(* CODESYS project native.xml

Project tree, tasks and I/O mapping:
  Device : CODESYS Control Win V3 x64, CODESYS, version 3.5.21.40
    application Application
      libraries: Standard, 3.5.18.0 (System)
      task MainTask (cyclic, interval t#20ms, priority 1) calls PLC_PRG
      data type E_SystemState
      global variables GVL_IO
      global variables GVL_System
      program PLC_PRG [ST]
*)

// Device/Application/E_SystemState
TYPE E_SystemState :
(
    STOPPED,
    IDLE_READY,
    WAIT_TRAY_EMPTY,
    TRANSFER,
    FAULT
);
END_TYPE

// Device/Application/GVL_IO
{attribute 'qualified_only'}
VAR_GLOBAL
	 (* Inputs *)
    PB_START       : BOOL;
    PB_STOP        : BOOL;
    PB_RESET       : BOOL;
    E_STOP_OK      : BOOL := TRUE;

    PE_INFEED      : BOOL;
    PE_CLEAR       : BOOL := TRUE;    (* often 'clear' is TRUE when not blocked *)

    ITEM_TYPE_A    : BOOL;            (* TRUE = route to Tray A *)
    TRAY_A_EMPTY   : BOOL := TRUE;
    TRAY_B_EMPTY   : BOOL := TRUE;

    (* Outputs *)
    MTR_RUN        : BOOL;
    DIVERT_TO_A    : BOOL;
    DIVERT_TO_B    : BOOL;
    ALARM          : BOOL;
END_VAR

// Device/Application/GVL_System
{attribute 'qualified_only'}
VAR_GLOBAL
	State			: E_SystemState := STOPPED;
	NextState		: E_SystemState := STOPPED;
	
	RouteToA     : BOOL;          (* latched route for current item *)
    RouteLatched : BOOL := FALSE; (* true once route is captured *)
    FaultLatched : BOOL := FALSE;

    Prev_PE_Clear : BOOL := TRUE; (* for edge detect *)
END_VAR

// Device/Application/PLC_PRG
PROGRAM PLC_PRG
VAR
	  clear_rise : BOOL;
END_VAR

(* Default: remain in current state *)
GVL_System.NextState := GVL_System.State;

(* Rising edge when PE_CLEAR goes from 0 -> 1 (blocked -> clear) *)
clear_rise := (NOT GVL_System.Prev_PE_Clear) AND (GVL_IO.PE_CLEAR);
GVL_System.Prev_PE_Clear := GVL_IO.PE_CLEAR;

(* Default outputs: safe *)
GVL_IO.MTR_RUN := FALSE;
GVL_IO.DIVERT_TO_A := FALSE;
GVL_IO.DIVERT_TO_B := FALSE;
GVL_IO.ALARM := FALSE;

(* E-stop fault: immediate, latched *)
IF NOT GVL_IO.E_STOP_OK THEN
    GVL_System.FaultLatched := TRUE;
    GVL_System.State := FAULT;
    RETURN;
END_IF;

CASE GVL_System.State OF

STOPPED:
    (* System is safe, waiting for start *)
	
	GVL_System.RouteLatched := FALSE;
	
    IF GVL_IO.PB_START AND NOT GVL_System.FaultLatched THEN
        GVL_System.NextState := IDLE_READY;
    END_IF;

IDLE_READY:
    (* waiting for item *)
    IF GVL_IO.PE_INFEED THEN
        GVL_System.NextState := WAIT_TRAY_EMPTY;
    END_IF;

WAIT_TRAY_EMPTY:
    (* Latch route once per item *)
    IF NOT GVL_System.RouteLatched THEN
        GVL_System.RouteToA := GVL_IO.ITEM_TYPE_A;   (* TRUE=A, FALSE=B *)
        GVL_System.RouteLatched := TRUE;
    END_IF;

    (* Wait until destination tray is empty *)
    IF GVL_System.RouteToA THEN
        (* Route A *)
        IF GVL_IO.TRAY_A_EMPTY THEN
            GVL_System.NextState := TRANSFER;
        END_IF;
    ELSE
        (* Route B *)
        IF GVL_IO.TRAY_B_EMPTY THEN
            GVL_System.NextState := TRANSFER;
        END_IF;
    END_IF;

TRANSFER:
    (* Command diverter to latched route *)
    IF GVL_System.RouteToA THEN
        GVL_IO.DIVERT_TO_A := TRUE;
    ELSE
        GVL_IO.DIVERT_TO_B := TRUE;
    END_IF;

    (* Run conveyor *)
    GVL_IO.MTR_RUN := TRUE;

    (* Stop transfer when item clears the zone *)
    IF clear_rise THEN
        GVL_IO.MTR_RUN := FALSE;
        GVL_System.RouteLatched := FALSE;     (* ready for next item *)
        GVL_System.NextState := IDLE_READY;
    END_IF;

FAULT:
    GVL_IO.ALARM := TRUE;
    IF GVL_IO.PB_RESET AND GVL_IO.E_STOP_OK THEN
        GVL_System.FaultLatched := FALSE;
        GVL_System.RouteLatched := FALSE;
        GVL_System.NextState := STOPPED;
    END_IF;

END_CASE;

(* State update *)
GVL_System.State := GVL_System.NextState;

END_PROGRAM
